PROGRAM MAIN_Fast
VAR
END_VAR

(*
The SerialLineControl function block is supposed to be called in every PLC cycle.
It communicates with the serial line hardware device and transmits or receives data.
The SerialLineControl can be called in the standard task (e.g.for PcCOM port usage) 
or in a separate fast task (e.g.for terminal usage) as well.
A fast separate task will be necessary at high baud rates or with KL6001 terminals 
which have a small process image (3 or 5 data bytes only)
*)

(* background communication with the EL6001 terminal *)
BackgroundEL();

END_PROGRAM

(* stored: Version 1.1.0.1, ProductVersion 3.1.4024.9
   POU MAIN_Fast: Id {5f28e37e-dc10-4a87-9cb9-19052eeb3568}, SpecialFunc None *)
